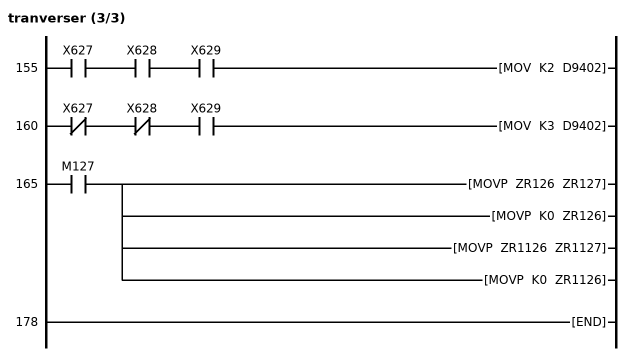
[picture p288: ladder of tranverser, rungs at steps 155 to 178]
155   LD      X627
      AND     X628
      AND     X629
      MOV     K2 D9402
160   LDI     X627
      ANI     X628
      AND     X629
      MOV     K3 D9402
165   LD      M127
      MOVP    ZR126 ZR127
      MOVP    K0 ZR126
      MOVP    ZR1126 ZR1127
      MOVP    K0 ZR1126
178   END
END_PROGRAM

PROGRAM unload
0     END
END_PROGRAM

PROGRAM x-lift
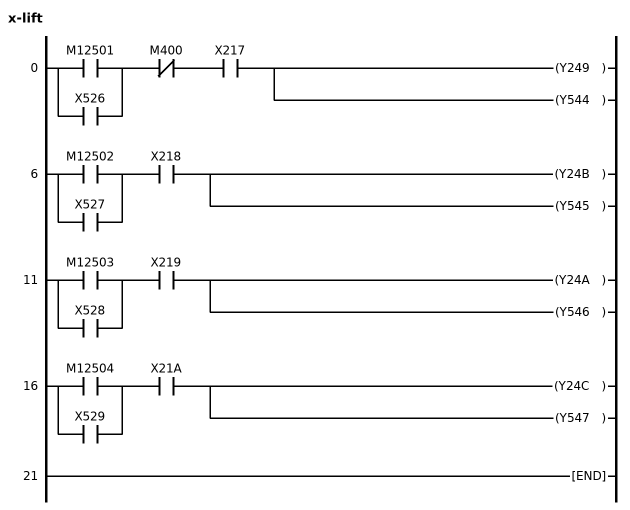
0     LD      M12501
      OR      X526
      ANI     M400
      AND     X217
      OUT     Y249
      OUT     Y544
6     LD      M12502
      OR      X527
      AND     X218
      OUT     Y24B
      OUT     Y545
11    LD      M12503
      OR      X528
      AND     X219
      OUT     Y24A
      OUT     Y546
16    LD      M12504
      OR      X529
      AND     X21A
      OUT     Y24C
      OUT     Y547
21    END
END_PROGRAM
